{attribute 'hide_all_locals'}
FUNCTION_BLOCK EcMasterState IMPLEMENTS IEcTask
VAR_INPUT
END_VAR
VAR_OUTPUT
END_VAR
VAR
	iState : INT;
	getMasterState : Tc2_EtherCAT.FB_EcGetMasterState;
	_execute: BOOL;
	_done: BOOL;
	_busy: BOOL;
	_error: BOOL;
	
END_VAR

CASE iState OF
	0:
		IF _execute THEN
			_done := FALSE;
			_busy := TRUE;
			_error := FALSE;
			getMasterState.bExecute := TRUE;
			IF getMasterState.bBusy THEN
				iState := 10;
				_execute := false;
			END_IF
		END_IF
	10:
		IF NOT getMasterState.bBusy THEN
			IF NOT getMasterState.bError THEN
				_done := TRUE;
			ELSE
				_error := TRUE;
			END_IF
			_busy := FALSE;
			getMasterState.bExecute := FALSE;
			iState := 0;
		END_IF
END_CASE

getMasterState(sNetId := Tc2_System.F_CreateAmsNetId(nIds := NetId));

{warning 'add method implementation '}
METHOD Abort : BOOL
getMasterState.bExecute := FALSE;
_busy := FALSE;
_execute := FALSE;
Abort := TRUE;
iState := 0;
END_METHOD

{warning 'add property implementation'}
PROPERTY Busy : BOOL
GET
Busy := _busy;
END_GET
END_PROPERTY

{warning 'add property implementation'}
PROPERTY Done : BOOL
GET
Done := _done;
END_GET
END_PROPERTY

{warning 'add property implementation'}
PROPERTY Error : BOOL
GET
Error := _error;
END_GET
END_PROPERTY

{warning 'add method implementation '}
METHOD Execute : BOOL
IF NOT getMasterState.bBusy THEN
	Execute := _execute := TRUE;
END_IF
END_METHOD

PROPERTY MasterState : word
GET
MasterState := getMasterState.state;
END_GET
END_PROPERTY

{warning 'add property implementation'}
PROPERTY NetID : amsnetid
GET
NetID := _netId;
END_GET
SET
_netId := NetID;
END_SET
END_PROPERTY

END_FUNCTION_BLOCK

(* stored: Version 1.1.0.1, ProductVersion 3.1.4024.9
   POU EcMasterState: Id {6636f90e-bd69-4e56-ba7e-95eafcef2973}, SpecialFunc None
   Method Abort: Id {29c6c77b-7079-4478-9fc0-6055e95e6e54}
   Property Busy: Id {50b11319-8e0f-46b7-ad99-a3ac18cd5a6a}
   Get Get: Id {c4b66164-e6ea-479c-bb28-d8869b1dce87}
   Property Done: Id {14930a58-c42f-459a-ab64-04ed546453ef}
   Get Get: Id {2412ef48-df64-47c3-a2c5-3ee43e77d52c}
   Property Error: Id {8d052741-b46a-406f-b65b-753707a76019}
   Get Get: Id {4f14d53c-9e31-48d9-b645-9767a1b80fd6}
   Method Execute: Id {f339eb4e-92ce-40a5-9935-97fc771e677a}
   Property MasterState: Id {b72b5599-8b4f-4684-9b6e-402b7ef6f94c}
   Get Get: Id {a6ab4d4c-33e9-4ff3-9638-a2f1014bd285}
   Property NetID: Id {8b8a36e2-e0d0-4fd8-89c8-10e431334d51}
   Get Get: Id {5442ff03-8004-4a83-a3b2-d137aa865efd}
   Set Set: Id {761843ad-5811-47ad-bf08-0c885c7cc268} *)
